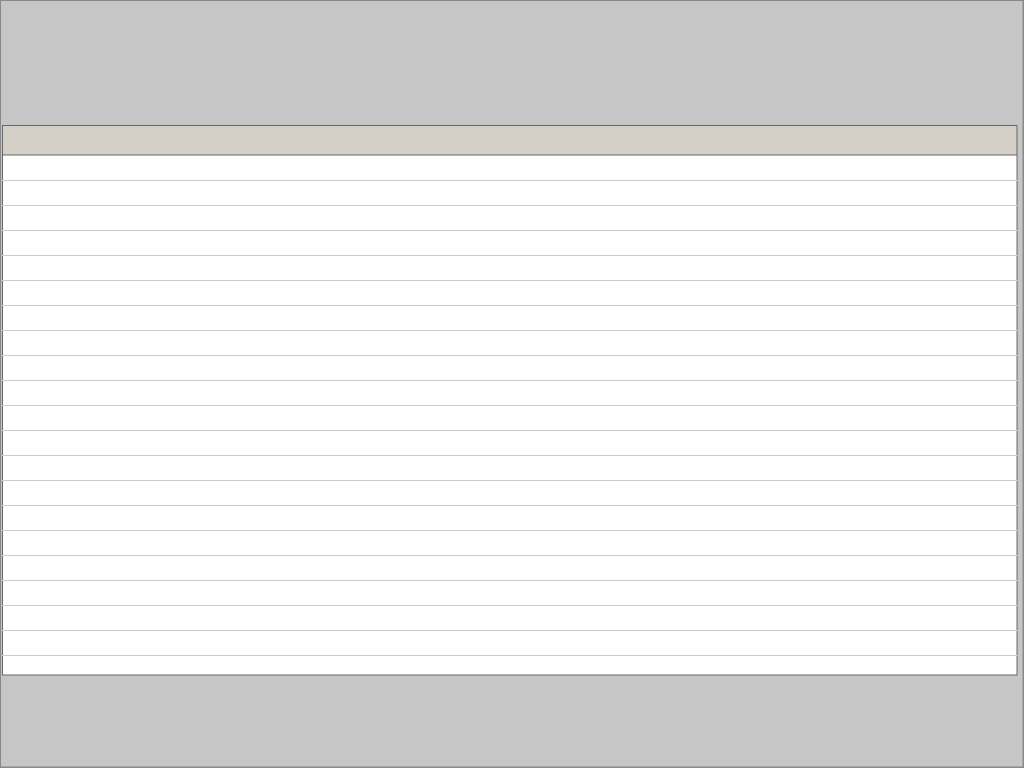
VISUALIZATION SS_12_AlarmsTests  // 1024x768
    Frame (0,0 1024x768)
        shows SS_91_Template(header := gHMIData.hmiHeader)
    Table (2,125 1015x550), data array: gmsgTest.msgArry
        p3854506369: gmsgTest.msgArry[INDEX].timeRaised
        p1892666644: gmsgTest.msgArry[INDEX].timeResolved
        p338671338: gmsgTest.msgArry[INDEX].text
        p2170511999: gmsgTest.msgArry[INDEX].source
        p2232123230: Time Raised
        p511219082: Time Resolved
        p1755163831: Message
        p4092479075: Location
        Columns.Column.[0].Template: gmsgTest.msgArryStyle[INDEX].isColoured; gmsgTest.msgArryStyle[INDEX].colourToApply
        Columns.Column.[1].Template: gmsgTest.msgArryStyle[INDEX].colourToApply; gmsgTest.msgArryStyle[INDEX].isColoured
        Columns.Column.[2].Template: gmsgTest.msgArryStyle[INDEX].isColoured; gmsgTest.msgArryStyle[INDEX].colourToApply
        Columns.Column.[3].Template: gmsgTest.msgArryStyle[INDEX].colourToApply; gmsgTest.msgArryStyle[INDEX].isColoured
END_VISUALIZATION

(* stored: Version 1.1.0.1, ProductVersion 3.1.4024.12
   Visu SS_12_AlarmsTests: Id {f0caa955-e950-4402-b6fa-6d4c00190f55} *)
